FUNCTION_BLOCK FB_SEL_COLOR (* COLOR Selection *)
  (* Standard: 61499-1 *)
  (* Version 0.1, 2004-06-21, JHC, Rockwell Automation, Moved from hmi to math. *)
  (* Version 0.0, 2001-04-05, JHC, Rockwell Automation, First XML version. *)
  (* Compiler header: package fb.rt.math; *)
  (* Compiler Java Sun JDK 1.4.2 *)
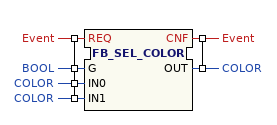
  EVENT_INPUT
    REQ WITH G, IN0, IN1;
  END_EVENT
  EVENT_OUTPUT
    CNF WITH OUT;
  END_EVENT
  VAR_INPUT
    G : BOOL; (* Selector *)
    IN0 : COLOR; (* Selected when G=0 *)
    IN1 : COLOR; (* Selected when G=1 *)
  END_VAR
  VAR_OUTPUT
    OUT : COLOR; (* Selected value *)
  END_VAR
  ALGORITHM REQ IN JAVA:
public void service_REQ(boolean qi){
OUT.value=G.value?IN1.value:IN0.value;}
CNF.serviceEvent(this);}
  END_ALGORITHM
END_FUNCTION_BLOCK
